FUNCTION_BLOCK FB_LevitationSystem
VAR_INPUT
END_VAR
VAR_OUTPUT
	eCondition : eConditionCheck;
END_VAR
VAR
	eMode : eSystemMode;
END_VAR

PROPERTY setSLEEP : BOOL
SET
IF setSLEEP THEN
	eMode := eSystemMode.SLEEP;
ELSE
	eMode := eSystemMode.RUN;
END_IF
END_SET
END_PROPERTY

END_FUNCTION_BLOCK

(* stored: Version 1.1.0.1, ProductVersion 3.1.4024.12
   POU FB_LevitationSystem: Id {45b5dcec-3c1d-41ef-adf9-89d78336b527}, SpecialFunc None
   Property setSLEEP: Id {eddd6ec8-da5e-43f0-9778-e8a801acc406}
   Set Set: Id {2adcb4b0-dd81-47de-87f7-52be68cb2e7e} *)
